Staubli VAL3: Main.dtx

mdesc mNomSpeed
bool bExit
bool bUserRefresh
aio aAio
string sParameter
string sListItemValue
bool bListRefresh
string sPath
